(*

.. <legal notes>

legal notes
=================
| SPDX-FileCopyrightText: © 2025 Oleksandr Tiutyk <trofimich@gmail.com>
| SPDX-License-Identifier: LGPL-3.0-only
| For details check: LGPL-3.0-only_

.. _LGPL-3.0-only: https://www.gnu.org/licenses/lgpl-3.0.en.html

.. </legal notes>

*)

INTERFACE ITask EXTENDS IObject

{attribute 'monitoring' := 'call'}
{attribute 'OPC.UA.DA.Property' := '1'}
{attribute 'OPC.UA.DA.Access' := '1'}
PROPERTY Done : BOOL
GET
END_GET
END_PROPERTY

{attribute 'monitoring' := 'call'}
{attribute 'OPC.UA.DA.Property' := '1'}
{attribute 'OPC.UA.DA.Access' := '1'}
PROPERTY Error : BOOL
GET
END_GET
END_PROPERTY

{attribute 'monitoring' := 'call'}
{attribute 'OPC.UA.DA.Property' := '1'}
{attribute 'OPC.UA.DA.Access' := '1'}
PROPERTY ErrorMessage : REFERENCE TO ERROR_MESSAGE
GET
END_GET
END_PROPERTY

METHOD Execute
END_METHOD

{attribute 'monitoring' := 'call'}
{attribute 'OPC.UA.DA.Property' := '1'}
{attribute 'OPC.UA.DA.Access' := '1'}
PROPERTY Running : BOOL
GET
END_GET
END_PROPERTY

METHOD Start
END_METHOD

{attribute 'monitoring' := 'call'}
{attribute 'OPC.UA.DA.Property' := '1'}
{attribute 'OPC.UA.DA.Access' := '1'}
PROPERTY StateChanged : BOOL
GET
END_GET
END_PROPERTY

END_INTERFACE

(* stored: Version 1.1.0.1
   Itf ITask: Id {33cd9918-3d9c-4cce-bc0c-72399b027fa3}
   Property Done: Id {ef9f248d-3252-4ffa-aac3-0418e1335c37}
   Get Get: Id {dfaea843-6fb1-4dcb-81b1-47917a384f3e}
   Property Error: Id {7a16200e-ba54-400f-8eb2-30023de937d5}
   Get Get: Id {a77db7b9-68ef-4cc4-95b5-ec801cc3280a}
   Property ErrorMessage: Id {9ef08aa6-77e6-45e8-aed3-0a06698ec0ba}
   Get Get: Id {c1078902-43dd-41df-be38-e2e04eaaa7a1}
   Method Execute: Id {60763b55-6821-4e9a-af1a-388d0c4ba48c}
   Property Running: Id {0bf76d8b-a1ea-4fc4-9149-9ac96039509d}
   Get Get: Id {bdaaed50-6e12-4f03-ab47-242eb0c00668}
   Method Start: Id {aa1685c2-0469-4461-956f-0e59ffd4e8ec}
   Property StateChanged: Id {8a597cd6-7e06-467c-85ae-5adc9086e4f8}
   Get Get: Id {2fd6fc94-ba43-423a-af7b-e0bf9d2d1aac} *)
